// TIA Portal V20 export
DATA_BLOCK "PeaInformationLabel"   // DB5
TITLE = PeaInformationLabel
{ S7_Optimized_Access := 'TRUE' }
AUTHOR : Siemens AG
FAMILY : MTP
VERSION : 1.0
// List of product- and instance-specific information for the PEA handling within a modular plant environment.
// stored: InstanceOfName typeMTPPeaInformationLabel, InstanceOfType UDT
"typeMTPPeaInformationLabel"
   // VAR
   //    AssetId : String := 'CFL_POC';
   //    ComponentName : String := 'name';
   //    DeviceClass : String := 'class';
   //    DeviceHealth { ExternalWritable := 'False'} : Byte;
   //    DeviceManual { ExternalWritable := 'False'} : String := '0.1';
   //    DeviceRevision { ExternalWritable := 'False'} : String := '0.1';
   //    HardwareRevision { ExternalWritable := 'False'} : String := '0.1';
   //    Manufacturer { ExternalWritable := 'False'} : String := '0.1';
   //    ManufacturerUri { ExternalWritable := 'False'} : String := '0.1';
   //    Model { ExternalWritable := 'False'} : String := '0.1';
   //    ProductCode { ExternalWritable := 'False'} : String := '0.1';
   //    ProductInstanceUri { ExternalWritable := 'False'} : String := '0.1';
   //    RevisionCounter { ExternalWritable := 'False'} : Int;
   //    SerialNumber { ExternalWritable := 'False'} : String := '0001';
   //    SoftwareRevision { ExternalWritable := 'False'} : String := '0.1';
   // END_VAR
BEGIN
END_DATA_BLOCK
